FUNCTION F_ArraySum : INT
VAR_INPUT
	  aSample : ARRAY[1..3] OF INT;
	  
END_VAR
VAR
    n   : INT;
    nSum : INT := 0;
END_VAR

FOR n := 1 TO 3 DO
    nSum := nSum + aSample[n];
END_FOR

F_ArraySum := nSum;

END_FUNCTION

(* stored: Version 1.1.0.1, ProductVersion 3.1.4024.16
   POU F_ArraySum: Id {4e96d3f6-7a12-4212-939f-7ec0f0fec90f}, SpecialFunc None *)
